// TIA Portal V20 export
DATA_BLOCK "IdentRfHmi"   // DB213
// stored: MemoryReserve 100
   VAR
      unitIdentRf : Array[1.."NO_OF_UNITS"] of "typeEMIdentRf";
   END_VAR
BEGIN
END_DATA_BLOCK
